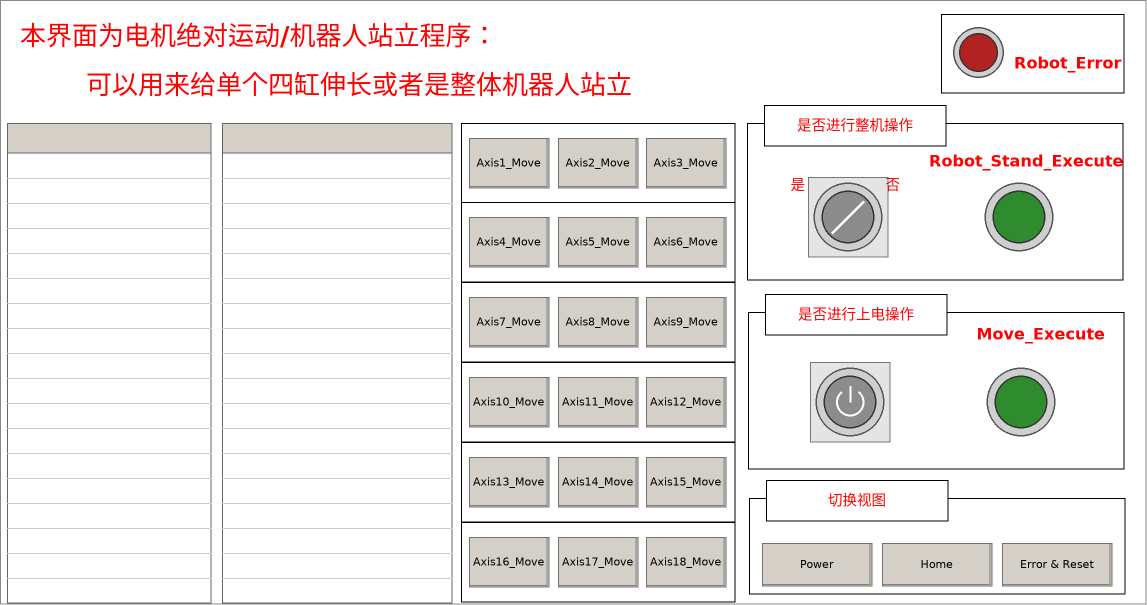
VISUALIZATION Visu_Walking_Robot_Stand  // 1147x605
    Rectangle (941,14 183x79)
    Rectangle (748,312 376x157)
    Label (964,318 154x32), "Move_Execute"
    Rectangle (765,294 182x41), "是否进行上电操作"
    Lamp1 (981,362 80x80), variable: Walking_Robot_Control.Move_Execute, style: Lamp-Lamp1-Green
    PowerSwitch (810,362 80x80), variable: Walking_Robot_Control.Move_Execute, behaviour: TOGGLE, style: Switch-PowerSwitch-Gray
    Lamp1 (948,23 61x59), variable: Walking_Robot_Control.Robot_Error, style: Lamp-Lamp1-Red
    Label (17,15 597x42), "本界面为电机绝对运动/机器人站立程序："
    Label (83,64 719x42), "可以用来给单个四缸伸长或者是整体机器人站立"
    Rectangle (747,123 376x157)
    Rectangle (764,105 182x41), "是否进行整机操作"
    Lamp1 (979,177 80x80), variable: Walking_Robot_Control.Robot_Stand_Execute, style: Lamp-Lamp1-Green
    RotarySwitch (808,177 80x80), variable: Walking_Robot_Control.Robot_Stand_Execute, behaviour: TOGGLE, style: Switch-RotarySwitch-Gray
    Label (863,170 60x30), "否"
    Label (768,170 60x30), "是"
    Label (991,47 154x32), "Robot_Error"
    Table (7,123 204x480), data array: Walking_Robot_Control.Axis_ActPostion
        p3854506369: Walking_Robot_Control.Axis_ActPostion[INDEX]
    Table (222,123 230x480), data array: Walking_Robot_Control.MoveAbsoluteDone
        p3854506369: Walking_Robot_Control.MoveAbsoluteDone[INDEX]
    Rectangle (461,123 274x80)
    Button (469,138 80x50), "Axis1_Move"
        toggle Walking_Robot_Control.Axis_Absolute_Eable[1]
    Button (646,138 80x50), "Axis3_Move"
        toggle Walking_Robot_Control.Axis_Absolute_Eable[3]
    Button (558,138 80x50), "Axis2_Move"
        toggle Walking_Robot_Control.Axis_Absolute_Eable[2]
    Rectangle (461,202 274x80)
    Button (469,217 80x50), "Axis4_Move"
        toggle Walking_Robot_Control.Axis_Absolute_Eable[4]
    Button (646,217 80x50), "Axis6_Move"
        toggle Walking_Robot_Control.Axis_Absolute_Eable[6]
    Button (558,217 80x50), "Axis5_Move"
        toggle Walking_Robot_Control.Axis_Absolute_Eable[5]
    Rectangle (461,282 274x80)
    Button (469,297 80x50), "Axis7_Move"
        toggle Walking_Robot_Control.Axis_Absolute_Eable[7]
    Button (646,297 80x50), "Axis9_Move"
        toggle Walking_Robot_Control.Axis_Absolute_Eable[9]
    Button (558,297 80x50), "Axis8_Move"
        toggle Walking_Robot_Control.Axis_Absolute_Eable[8]
    Rectangle (461,362 274x80)
    Button (469,377 80x50), "Axis10_Move"
        toggle Walking_Robot_Control.Axis_Absolute_Eable[10]
    Button (646,377 80x50), "Axis12_Move"
        toggle Walking_Robot_Control.Axis_Absolute_Eable[12]
    Button (558,377 80x50), "Axis11_Move"
        toggle Walking_Robot_Control.Axis_Absolute_Eable[11]
    Rectangle (461,442 274x80)
    Button (469,457 80x50), "Axis13_Move"
        toggle Walking_Robot_Control.Axis_Absolute_Eable[13]
    Button (646,457 80x50), "Axis15_Move"
        toggle Walking_Robot_Control.Axis_Absolute_Eable[15]
    Button (558,457 80x50), "Axis14_Move"
        toggle Walking_Robot_Control.Axis_Absolute_Eable[14]
    Rectangle (461,522 274x80)
    Button (469,537 80x50), "Axis16_Move"
        toggle Walking_Robot_Control.Axis_Absolute_Eable[16]
    Button (646,537 80x50), "Axis18_Move"
        toggle Walking_Robot_Control.Axis_Absolute_Eable[18]
    Button (558,537 80x50), "Axis17_Move"
        toggle Walking_Robot_Control.Axis_Absolute_Eable[17]
    Label (923,145 207x32), "Robot_Stand_Execute"
    Rectangle (749,498 376x96)
    Rectangle (766,480 182x41), "切换视图"
    Button (762,543 110x43), "Power"
        OnMouseClick: change screen: Visu_Power
    Button (1002,543 110x43), "Error & Reset"
        OnMouseClick: change screen: Visu_Reset
    Button (882,543 110x43), "Home"
        OnMouseClick: change screen: Visu_Home
END_VISUALIZATION

(* stored: Version 1.1.0.1, ProductVersion 3.1.4020.12
   Visu Visu_Walking_Robot_Stand: Id {7a1ff3cc-fdc9-4f0b-b540-0d0cc169a48a} *)
